FUNCTION_BLOCK PnPVacuum (* Vacuum model *)
  (* Standard: 61499-2 *)
  (* Version 1.0, 2008-11-09, Cheng Pang, The University of Auckland, Stable build. *)
  (* Compiler header: package fb.rt.pnp; *)
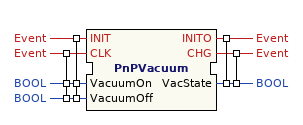
  EVENT_INPUT
    INIT WITH VacuumOn, VacuumOff; (* Initialization Request *)
    CLK WITH VacuumOn, VacuumOff; (* Clock signal *)
  END_EVENT
  EVENT_OUTPUT
    INITO WITH VacState; (* Initialization Confirm *)
    CHG WITH VacState; (* Execution Confirmation *)
  END_EVENT
  VAR_INPUT
    VacuumOn : BOOL; (* Input event qualifier *)
    VacuumOff : BOOL;
  END_VAR
  VAR_OUTPUT
    VacState : BOOL; (* State of vacuum *)
  END_VAR
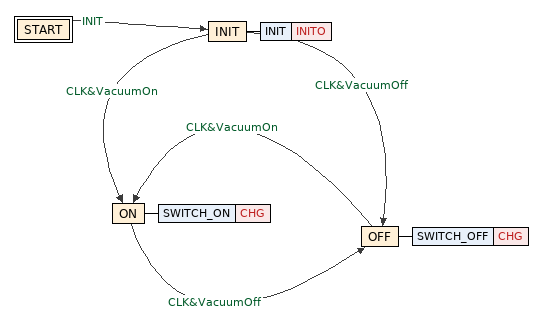
  EC_STATES
    START; (* Initial State *)
    INIT : INIT -> INITO; (* Initialization *)
    ON : SWITCH_ON -> CHG; (* Normal execution *)
    OFF : SWITCH_OFF -> CHG;
  END_STATES
  EC_TRANSITIONS
    START TO INIT := INIT;
    INIT TO OFF := CLK&VacuumOff;
    OFF TO ON := CLK&VacuumOn;
    ON TO OFF := CLK&VacuumOff;
    INIT TO ON := CLK&VacuumOn;
  END_TRANSITIONS
  ALGORITHM INIT IN Java: (* Initialization algorithm *)
//System.out.println("\n Vacuum.INIT:");
if(VacuumOn.value){
  VacState.value = true;
}
else if(VacuumOff.value){
  VacState.value = false;
}
//System.out.println("");
  END_ALGORITHM
  ALGORITHM SWITCH_ON IN Java:
VacState.value = true;
  END_ALGORITHM
  ALGORITHM SWITCH_OFF IN Java:
VacState.value = false;
  END_ALGORITHM
END_FUNCTION_BLOCK
